PROGRAM MAIN_FastAsPossible_ITc
VAR
	
	fbRtmode : FB_RtMode; 
	state : INT := 0;	
	bStart : BOOL; 
	hr: HRESULT;
	eCurrentMode: E_RtMode;
END_VAR


VAR_OUTPUT 
	value AT %Q* : UDINT;	
END_VAR

hr := fbrtmode.ip.GetTickMode(eCurrentMode);

CASE state OF
	0:
		IF(bStart = TRUE) THEN 		
			state:= 1;
			value:=100; // steps to decrement as Cyclic 
		END_IF
	1:
		IF(eCurrentMode = E_RtMode.RtMode_Cyclic) THEN 
			value:=value-1; //decrementing Cyclic (near realtime speed) 
			IF value = 0 THEN
				state := 2;
				value:=100000; // Steps to decrement as a FastAsPossible 						
				(*switch to fastaspossible mode*)			
				fbRtmode.ip.ChangeTickMode(E_RtMode.RtMode_FastAsPossible);
			END_IF 	
		ELSE 
			state := 98; // ERROR 
		END_IF
	2:
		IF(eCurrentMode = E_RtMode.RtMode_FastAsPossible) THEN 
			value:=value-1; //decrementing as fast as possible 
			IF value = 0 THEN
				(*switch back to cyclic mode*)			
				state := 0;
				fbRtmode.ip.ChangeTickMode(E_RtMode.RtMode_Cyclic);			
			END_IF
		ELSE 
			state := 99; // ERROR 
		END_IF
END_CASE

END_PROGRAM

(* stored: Version 1.1.0.1, ProductVersion 3.1.4025.18
   POU MAIN_FastAsPossible_ITc: Id {afd9ca21-21e0-4cf9-86ce-293511cbda74}, SpecialFunc None *)
